RoboDK station: EX_1_PICK_AND_PLACE.rdk

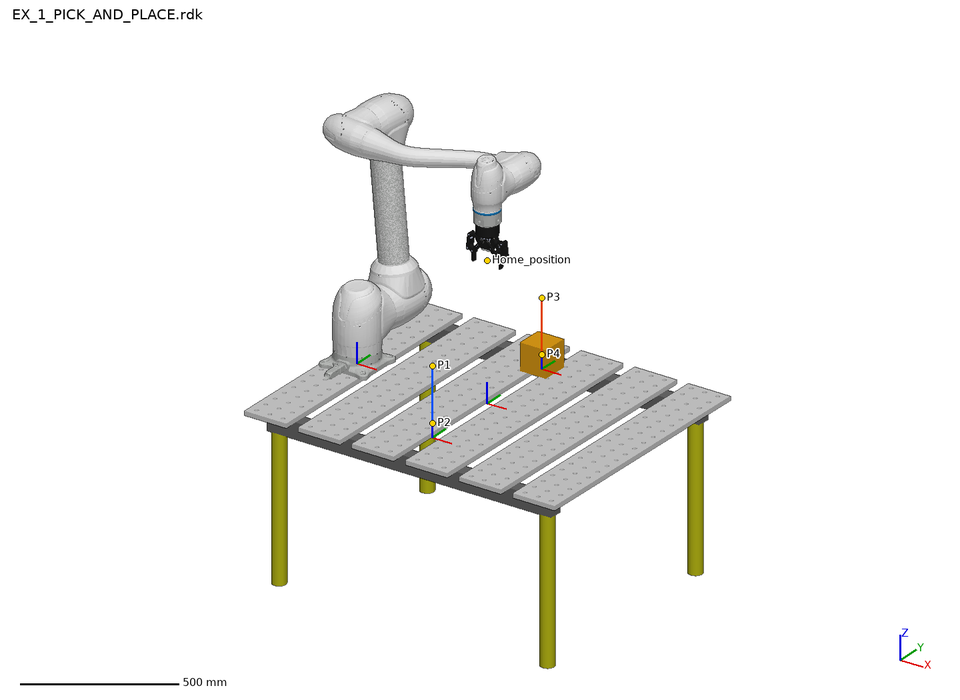
[picture v0: the station drawn from its stored meshes, robots at their saved joint values, targets as dots, program paths as lines]
Station EX_1_PICK_AND_PLACE (saved by RoboDK 5.8.0). Poses are relative to the parent item; angles as X-Y-Z fixed-axis rotations.
  - frame Doosan Robotics M1013 White Base at (-500, 0, 0) mm
    - robot Doosan Robotics M1013 White: 6 axes, payload 10 kg, reach 1300 mm, repeatability 0.05 mm, weight 33 kg
        modified DH rows (alpha deg, a mm, theta deg, d mm): 0, 0, 0, 152.5; -90, 0, -90, -34.506; 0, 620, -90, 0; -90, 0, 0, 559; 90, 0, 0, 0; -90, 0, 180, 121
        base shift (0, 0, 0) mm, rotated rx 0 ry 0 rz 180 deg
        joint limits [-360, -360, -160, -360, -360, -360] to [360, 360, 160, 360, 360, 360]; home [0, 0, 90, 0, 0, 0]; saved at [-3.957, -5.543, 97.449, 0, 88.093, -3.957]
      - tool RobotiQ 2F-85 Gripper (Open), TCP at (0, 0, 130) mm, size 147.4 x 75 x 146.8 mm
  - frame Base at (0, 0, 0) mm
    - object Table 1200x1000mm (Welding) at (0, 0, 0) mm, size 1193.8 x 965.2 x 609.6 mm, geometry from Table-1200x1000mm-Welding.sld
    - target Home_position (Cartesian target) at (0, 0, 500) mm, rotated rx -180 ry 0 rz -180 deg; joints [-3.957, -5.543, 97.449, 0, 88.093, -3.957] of Doosan Robotics M1013 White
  - frame Part_1 at (0, -300, 0) mm
    - target P1 (Cartesian target) at (0, 0, 250) mm, rotated rx -180 ry 0 rz -180 deg; joints [-34.356, 8.333, 109.96, 0, 61.707, -34.356] of Doosan Robotics M1013 White
    - target P2 (Cartesian target) at (0, 0, 50) mm, rotated rx -180 ry 0 rz -180 deg; joints [-34.356, 21.209, 118.997, 0, 39.794, -34.356] of Doosan Robotics M1013 White
  - frame Part_2 at (0, 300, 0) mm
    - target P3 (Cartesian target) at (0, 0, 250) mm, rotated rx 180 ry 0 rz -180 deg; joints [27.571, 8.333, 109.96, 0, 61.707, 27.571] of Doosan Robotics M1013 White
    - target P4 (Cartesian target) at (0, 0, 50) mm, rotated rx 180 ry 0 rz -180 deg; joints [27.571, 21.209, 118.997, 0, 39.794, 27.571] of Doosan Robotics M1013 White
    - object Cube 100mm at (-50, -50, 0) mm, size 100 x 100 x 100 mm, geometry from Cube-100mm.sld
  - program Reset_position (4 instructions, listed below)
  - program Picking (6 instructions, listed below)
  - program Placing (6 instructions, listed below)
  - program Main_program (7 instructions, listed below)
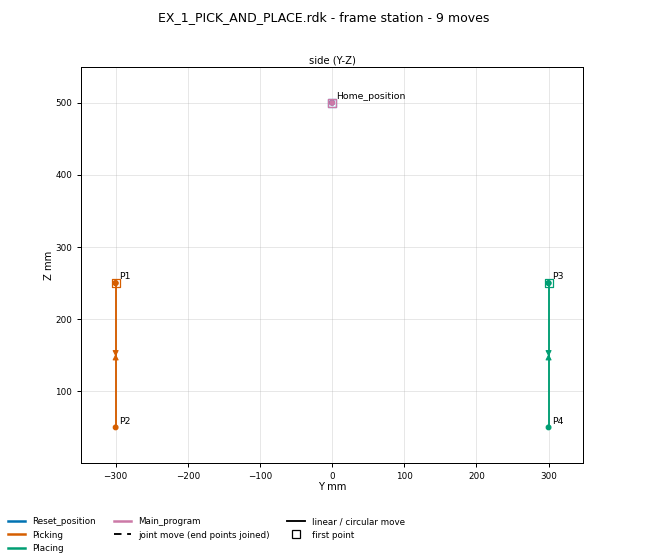
[picture p0: tool path of EX_1_PICK_AND_PLACE.rdk in frame station, 9 of 9 moves have a stored position in this frame; points joined in program order, loops and branches not executed]

--- program Reset_position (robot Doosan Robotics M1013 White) ---
  Set Ref.: Base
  Set Tool: RobotiQ 2F-85 Gripper (Open)
  Replace objects
  MoveJ (Home_position)

--- program Picking (robot Doosan Robotics M1013 White) ---
  Set Ref.: Part_1
  Set Tool: RobotiQ 2F-85 Gripper (Open)
  MoveJ (P1)
  MoveL (P2)
  Attach to RobotiQ 2F-85 Gripper (Open)
  MoveL (P1)

--- program Placing (robot Doosan Robotics M1013 White) ---
  Set Ref.: Part_2
  Set Tool: RobotiQ 2F-85 Gripper (Open)
  MoveJ (P3)
  MoveL (P4)
  Detach from RobotiQ 2F-85 Gripper (Open)
  MoveL (P3)

--- program Main_program (robot Doosan Robotics M1013 White) ---
  Set Ref.: Base
  Set Tool: RobotiQ 2F-85 Gripper (Open)
  MoveJ (Home_position)
  Call Picking
  Call Placing
  Set Ref.: Base
  MoveJ (Home_position)
